PROGRAM Systemauswertung
VAR
	Auswertung_R1		:FB_Auswertung;
	Auswertung_R2		:FB_Auswertung;
END_VAR

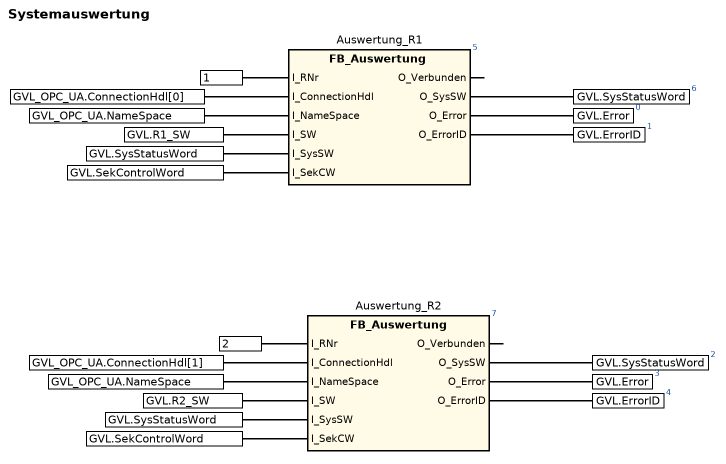
GVL.Error := Auswertung_R1.O_Error;
GVL.ErrorID := Auswertung_R1.O_ErrorID;
GVL.SysStatusWord := Auswertung_R2.O_SysSW;
GVL.Error := Auswertung_R2.O_Error;
GVL.ErrorID := Auswertung_R2.O_ErrorID;
Auswertung_R1(
    I_RNr := 1,
    I_ConnectionHdl := GVL_OPC_UA.ConnectionHdl[0],
    I_NameSpace := GVL_OPC_UA.NameSpace,
    I_SW := GVL.R1_SW,
    I_SysSW := GVL.SysStatusWord,
    I_SekCW := GVL.SekControlWord); // FB_Auswertung
GVL.SysStatusWord := Auswertung_R1.O_SysSW;
Auswertung_R2(
    I_RNr := 2,
    I_ConnectionHdl := GVL_OPC_UA.ConnectionHdl[1],
    I_NameSpace := GVL_OPC_UA.NameSpace,
    I_SW := GVL.R2_SW,
    I_SysSW := GVL.SysStatusWord,
    I_SekCW := GVL.SekControlWord); // FB_Auswertung

END_PROGRAM

(* stored: Version 1.1.0.1, ProductVersion 3.1.4024.12
   POU Systemauswertung: Id {0e713e24-ee02-460f-85c3-ce9c05c7a3ac}, SpecialFunc None *)
